TYPE ONE_BIT :
STRUCT
	e1 : BIT;
END_STRUCT
END_TYPE

(* stored: Version 1.1.0.1, ProductVersion 3.1.4024.11
   DUT ONE_BIT: Id {3095daaa-1d5e-44cd-93ec-6150e8d9b1f6} *)
